(* CODESYS project zadanie 3 sprawko3.project

Project tree, tasks and I/O mapping:
  Device : CODESYS Control Win V3, CODESYS, version 3.5.20.30
    application Application
      libraries: Standard, 3.5.18.0 (System)
      task VISU_TASK (cyclic, interval 100 ms, priority 31) calls VisuElems.Visu_Prg
      task MainTask (cyclic, interval t#20ms, priority 1) calls PLC_PRG_GK
      visualisation Visualization
      program PLC_PRG_GK [LD]
  libraries: Standard, 3.5.18.0 (System); VisuElemBase, * (System)
  text list GlobalTextList
*)

// Device/Application/PLC_PRG_GK
PROGRAM PLC_PRG_GK
VAR
    S1_GK, S2_GK, S3_GK: BOOL;
    S1_mono_GK, S1_bi_GK, S2_mono_GK, S2_bi_GK, S3_mono_GK, S3_bi_GK: BOOL;
    H1_GK, H2_GK, H3_GK: BOOL;
    H4_GK, H5_GK, H6_GK: BOOL;
 	instancjaRS: RS;
	TON_GK: TON;
	TOF_GK: TOF;
	TP_GK: TP;
	TONn_GK: TON;
END_VAR

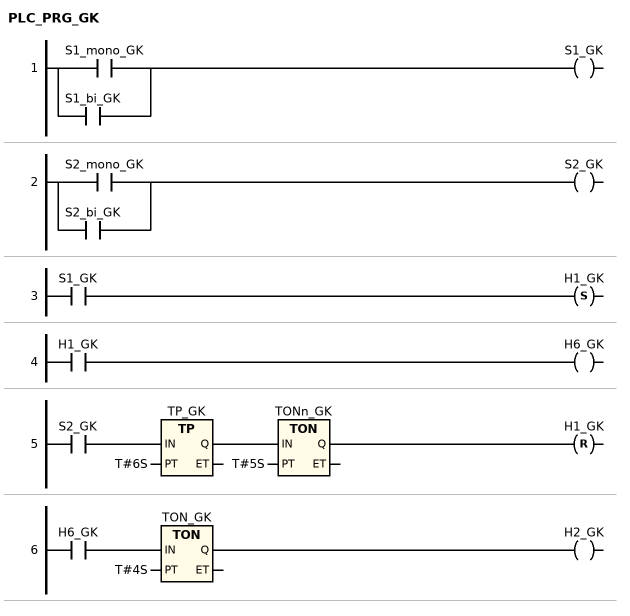
// NETWORK 1
S1_GK := S1_mono_GK OR S1_bi_GK;

// NETWORK 2
S2_GK := S2_mono_GK OR S2_bi_GK;

// NETWORK 3
H1_GK S= S1_GK;

// NETWORK 4
H6_GK := H1_GK;

// NETWORK 5
TP_GK(IN := S2_GK, PT := T#6S); // TP
TONn_GK(IN := TP_GK.Q, PT := T#5S); // TON
H1_GK R= TONn_GK.Q;

// NETWORK 6
TON_GK(IN := H6_GK, PT := T#4S); // TON
H2_GK := TON_GK.Q;

END_PROGRAM

// Device/Application/Visualization
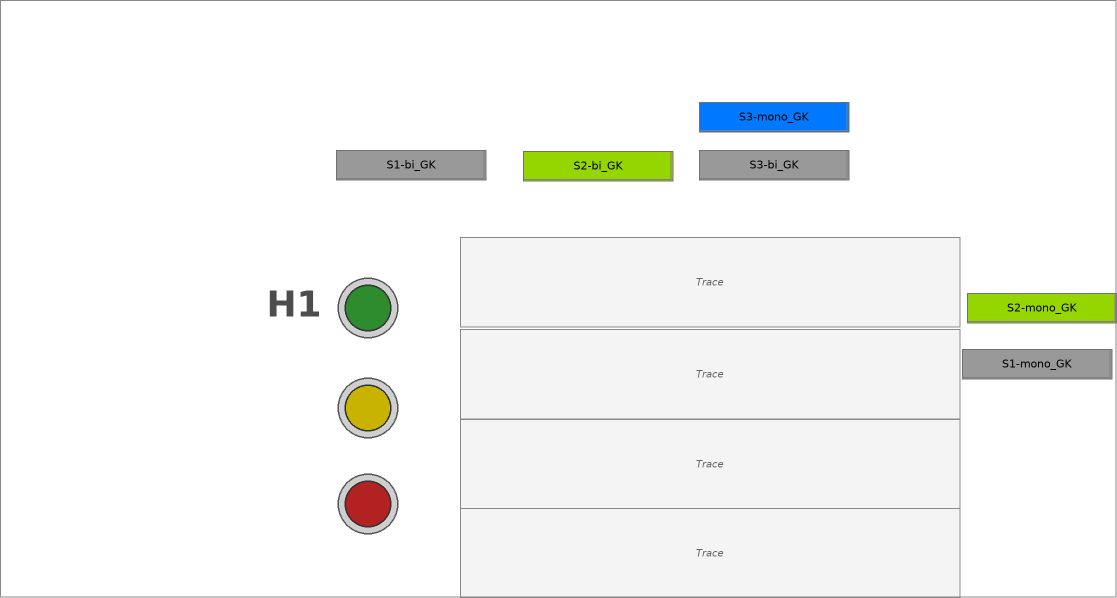
VISUALIZATION Visualization  // 1117x598
    Lamp1 (333,273 70x70), variable: PLC_PRG_GK.H1_GK, style: Lamp-Lamp1-Green
    Lamp1 (333,373 70x70), variable: PLC_PRG_GK.H2_GK, style: Lamp-Lamp1-Yellow
    Lamp1 (333,469 70x70), variable: PLC_PRG_GK.H3_GK, style: Lamp-Lamp1-Red
    Button (962,349 150x30), "S1-mono_GK"
        tap PLC_PRG_GK.S1_mono_GK
    Button (967,293 150x30), "S2-mono_GK"
        tap PLC_PRG_GK.S2_mono_GK
    Button (336,150 150x30), "S1-bi_GK"
        toggle PLC_PRG_GK.S1_bi_GK
    Button (523,151 150x30), "S2-bi_GK"
        toggle PLC_PRG_GK.S2_bi_GK
    Button (699,102 150x30), "S3-mono_GK"
        tap PLC_PRG_GK.S3_mono_GK
    Button (699,150 150x30), "S3-bi_GK"
        toggle PLC_PRG_GK.S3_bi_GK
    Trace (460,237 500x90)
    Label (219,289 150x30), "H1"
    Trace (460,329 500x90)
    Trace (460,419 500x90)
    Trace (460,508 500x90)
END_VISUALIZATION
